PROGRAM POU
VAR
	Mode: BOOL;
	Fan_speed: REAL;
	STATUS: BOOL;
	Manual: BOOL;
	Fan_0: FB_Fan;
	SETPOINT: REAL := 15;
	CURRNET: REAL := 10;
	STARTMAN: BOOL;
	STOPMAN: BOOL;
	STARTAUTO: BOOL;
	STOPAUTO: BOOL;
	EMERGSTOP: BOOL;
	FAULT: BOOL;
	CYCLERUN: BOOL;
	FAULT_LOG: STRING;
	DELAY_TIMER: TON;
	START_DELAY: TON;
	EMERGSTOP_STATUS: BOOL;
	BUZZER: BOOL;
	MODESELECT: INT;
	STOPDELAY: TIME;
	STARTDELAY: TIME;
	FB_SensorHandler_0: FB_SensorHandler;
	SESNORSTATUS: BOOL;
	INPUT: BOOL;
	OUTPUT: BOOL;
	FAULTSTATUS: STRING(50);
END_VAR

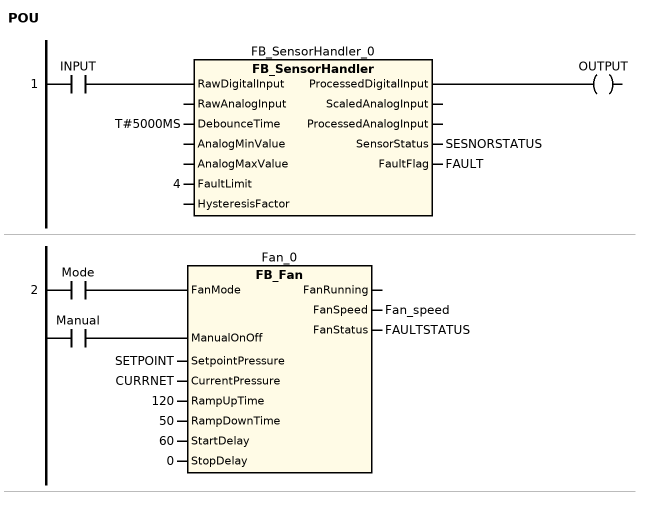
// NETWORK 1
FB_SensorHandler_0(
    RawDigitalInput := INPUT,
    DebounceTime := T#5000MS,
    FaultLimit := 4,
    SensorStatus => SESNORSTATUS,
    FaultFlag => FAULT); // FB_SensorHandler
OUTPUT := FB_SensorHandler_0.ProcessedDigitalInput;

// NETWORK 2
Fan_0(
    FanMode := Mode,
    ManualOnOff := Manual,
    SetpointPressure := SETPOINT,
    CurrentPressure := CURRNET,
    RampUpTime := 120,
    RampDownTime := 50,
    StartDelay := 60,
    StopDelay := 0,
    FanSpeed => Fan_speed,
    FanStatus => FAULTSTATUS); // FB_Fan

END_PROGRAM

(* stored: Version 1.1.0.1, ProductVersion 3.1.4024.13
   POU POU: Id {e229df73-6924-4730-af5d-bc0348d092d4}, SpecialFunc None *)
